PROGRAM MAIN
VAR
END_VAR

END_PROGRAM

(* stored: Version 1.1.0.1
   POU MAIN: Id {8811217b-2fd3-4514-b827-dcec12235d4b} *)
